PROGRAM MAIN
VAR
	
TimeStamper : NT_GetTime;
integer : INT;
mySQlsimulation : Array[1..100, 1..2]; 

END_VAR

END_PROGRAM

(* stored: Version 1.1.0.1, ProductVersion 3.1.4024.12
   POU MAIN: Id {507c972b-c2fd-445b-a16a-d48ecf9a24a3}, SpecialFunc None *)
